(* IEC 61131-3 sources: moqui-plc/iec61131/moqui/framework/src/main/org/moqui/device (part 2) *)

(* ---- ActuatorGroup.st ---- *)
(*
 * ActuatorGroup - demand-driven staging controller for up to ACTUATOR_GROUP_MAX_SIZE on/off actuators.
 *
 * Inspired by ABB ACH580 PFC (Pump and Fan Control, group 76. See ABB ACH580 drive firmware manual).
 * Progressively starts and stops Actuator FBs to match a varying process demand,
 * with automatic priority rotation (autochange) to balance accumulated run hours.
 *
 * Interface with Actuator FBs
 * The caller declares enableRequests and disableRequests arrays and wires them
 * to the VAR_IN_OUT inputs of each Actuator FB:
 *
 *   pump[i](enableRequest := enReq[i], disableRequest := disReq[i], ...);
 *   grp(enableRequests := enReq, disableRequests := disReq, ...);
 *
 * Both the Actuator and ActuatorGroup share the same array by reference (VAR_IN_OUT).
 * ActuatorGroup writes TRUE to issue a command;
 * the Actuator clears the flag to FALSE as its handshake acknowledgment.
 *
 * IMPORTANT: call each Actuator BEFORE ActuatorGroup in the PLC task so that
 * the actuatorEnabled feedback is current when ActuatorGroup evaluates it.
 *
 * Start / stop staging
 * startPoints[k] (k = 0..actuatorNum-1):
 *   While k actuators are running, if demandSetpoint > startPoints[k] continuously
 *   for startDelay, the next available actuator in the priority order is started (subject to runningNum < maxRunning).
 *   startPoints[0] is the threshold to start the very first actuator (0 -> 1).
 *
 * stopPoints[k] (k = 0..actuatorNum-2):
 *   While k+1 actuators are running, if demandSetpoint < stopPoints[k] continuously
 *   for stopDelay, the lowest-priority running actuator is stopped (subject to runningNum > minRunning).
 *   stopPoints[0] is the threshold to stop the last remaining actuator (1 -> 0).
 *
 * Demand must hold on one side of the threshold for the full delay before any action is taken.
 * Crossing back resets the timer (anti-cycling hysteresis).
 *
 * Fault / interlock recovery:
 *   Faulted or interlocked actuators are skipped during start selection.
 *   If a running actuator faults and runningNum drops below minRunning, the next
 *   available standby is started immediately (without waiting for startDelay).
 *
 * Autochange:
 * EvenWear: Rotate when the run-hour gap between any two non-faulted
 *           actuators exceeds maxWearImbalance AND demand <= autochangeLevel.
 *           The priority array is re-sorted by ascending runHours every cycle;
 *           a physical swap (stop most-used, start least-used) is
 *           triggered only when the imbalance threshold is exceeded.
 * FixedInterval: Rotate every autochangeInterval when demand <= autochangeLevel.
 * ExternalTrigger: Rotate on a rising edge of autochangeTrigger when demand <= autochangeLevel.
 * AllStopped: Rotate the index array whenever all actuators stop (group
 *             transitions to Disabled). No physical swap is needed because
 *             all are already stopped; the new order takes effect at the next group enable.
 *
 * Rotation sequence (EvenWear / FixedInterval / ExternalTrigger):
 *   1. Stop the selected actuator (disableRequest).
 *   2. Update the priority array (rotate or re-sort).
 *   3. Start the new highest-priority standby actuator (enableRequest).
 *   The group is in the Autochange FSM state for the duration of this sequence.
 *   runningNum briefly drops by 1; set minRunning = 0 if a momentary reduction
 *   is unacceptable and use process-side redundancy instead.
 *)
FUNCTION_BLOCK ActuatorGroup
	VAR_EXTERNAL CONSTANT
	    (*
		 * Maximum actuators supported. Array bounds in VAR_IN_OUT / VAR_INPUT
	     * must match this size exactly in the caller's declaration.
		 *)
	    ACTUATOR_GROUP_MAX_SIZE : UINT;
	END_VAR
	VAR_IN_OUT
	    (*
	     * Handshake arrays shared with the individual Actuator FBs.
	     * ActuatorGroup writes TRUE to command a start or stop.
	     * Each Actuator FB clears the flag to FALSE when it accepts the command.
	     *)
	    enableRequests : ARRAY[1..ACTUATOR_GROUP_MAX_SIZE] OF BOOL;
	    disableRequests : ARRAY[1..ACTUATOR_GROUP_MAX_SIZE] OF BOOL;
	END_VAR
	VAR_INPUT
		(* Actuator group metadata for logging purpose *)
		actuatorGroupId : STRING;
		actuatorGroupName : STRING;

	    (* Topology *)
	    (* Total actuators declared in the group. Must be 1..ACTUATOR_GROUP_MAX_SIZE. *)
	    actuatorNum : UINT := 1;
	    (* Minimum actuators to keep running simultaneously (0 = allow full stop). *)
	    minRunning : UINT := 1;
	    (* Maximum actuators allowed running simultaneously. *)
	    maxRunning : UINT := 1;

	    (* Process demand *)
	    (* Demand setpoint in percent (0.0 ... 100.0). Drives all start/stop decisions. *)
	    demandSetpoint : REAL;

	    (*
	     * Start / stop thresholds.
	     * startPoints[k]: demand level that triggers starting the (k+1)-th
	     * actuator while exactly k are currently running (k = 0..actuatorNum-1).
	     * startPoints[0] = threshold to start the first actuator (0 -> 1).
		 *)
	    startPoints : ARRAY[0..7] OF REAL;
	    (*
	     * stopPoints[k]: demand level below which the (k+1)-th running actuator is stopped (k = 0..actuatorNum-2).
	     * stopPoints[0] = threshold to stop the last actuator (1 -> 0).
	     *)
	    stopPoints : ARRAY[0..7] OF REAL;
	    (* Demand must stay above startPoints[k] for this long before a start. *)
	    startDelay : TIME := T#10s;
	    (* Demand must stay below stopPoints[k] for this long before a stop. *)
	    stopDelay : TIME := T#10s;

	    (* Autochange *)
	    autochange : ActuatorGroupAutochange := ActuatorGroupAutochange.None;
	    (* Period for FixedInterval rotation. *)
	    autochangeInterval : TIME := T#1h;
	    (*
	     * Max allowed run-hour gap between most-used and least-used actuator
	     * before EvenWear triggers a swap (hours, e.g. 72.0 for 3 days).
	     *)
	    maxWearImbalance : REAL := 72.0;
	    (* Autochange is only triggered when demandSignal <= autochangeLevel. *)
	    autochangeLevel : REAL := 100.0;
	    (* Rising edge triggers an immediate autochange (ExternalTrigger mode). *)
	    autochangeTrigger : BOOL;

	    (* Per-actuator feedback *)
	    (*
	     * Map actuatorEnabled[i] from Actuator[i].enable (TRUE in EnablePhase
	     * AND Enabled states - i.e., the actuator is active or starting up).
	     *)
	    actuatorEnabled : ARRAY[1..ACTUATOR_GROUP_MAX_SIZE] OF BOOL;
	    (* Map actuatorFault[i] from Actuator[i].fault. *)
	    actuatorFault : ARRAY[1..ACTUATOR_GROUP_MAX_SIZE] OF BOOL;
	    (* External maintenance / hardware interlock flag per actuator. *)
	    actuatorInterlocked : ARRAY[1..ACTUATOR_GROUP_MAX_SIZE] OF BOOL;
	    (* Cumulative run time in hours, maintained by the caller (e.g., a REAL counter incremented by 1/3600 each second). *)
	    runHours : ARRAY[1..ACTUATOR_GROUP_MAX_SIZE] OF REAL;

	    (* Group commands *)
	    (*
	      * Rising edge (FALSE->TRUE) starts the group (Disabled -> Running).
	      * Cleared by the FB when the transition is accepted.
	     *)
	    groupEnable : BOOL;
	    (*
	     * Rising edge (FALSE->TRUE) stops the group (Running -> Stopping -> Disabled).
	     * Cleared by the FB when the transition is accepted.
	     *)
	    groupDisable : BOOL;
	END_VAR
	VAR_OUTPUT
	    (* Current group FSM state. *)
	    status : ActuatorGroupStatus := ActuatorGroupStatus.Disabled;
	    (* Actuators neither faulted nor interlocked (available for use). *)
	    availableNum : UINT;
	    (* Actuators currently active (Enabled or EnablePhase). *)
	    runningNum : UINT;
	    (* TRUE when nAvailable < actuatorNum (one or more offline/faulted). *)
	    degraded : BOOL;
	    (* TRUE when a fault has left runningNum below minRunning. *)
	    underMinimum : BOOL;
	    (* TRUE when configuration inputs are invalid. *)
	    invalidConfig : BOOL;
	    (* TRUE while an autochange rotation is in progress. *)
	    autochangeActive : BOOL;
		(* Logger name for centralized signal management *)
		loggerName : STRING;
	END_VAR
	VAR
	    (* Internal FSM state *)
	    internalStatus : ActuatorGroupStatus := ActuatorGroupStatus.Disabled;

	    (* Priority order *)
	    (*
		 * sortedIdx[1] = first to start / last to stop.
	     * sortedIdx[actuatorNum] = last to start / first to stop.
	     * Initialised to [1, 2, … actuatorNum] on the first call.
	     *)
	    sortedIdx : ARRAY[1..ACTUATOR_GROUP_MAX_SIZE] OF UINT;

	    (* Autochange bookkeeping *)
	    autochangeStep : UINT; (* 0 = idle, 1 = stopping old, 2 = starting new *)
	    autochangeStopIdx : UINT; (* physical actuator slot being stopped *)
	    autochangeStartIdx : UINT; (* physical actuator slot being started *)
	    autochangeTrigOld : BOOL; (* previous cycle value for edge detection *)

	    (* Timer signals *)
	    (* Computed each cycle in the FSM; passed to TON FBs at the bottom. *)
	    startTimerTrig : BOOL;
	    stopTimerTrig : BOOL;
	    autochangeTimerTrig : BOOL;
	    startTimer : TON;
	    stopTimer : TON;
	    autochangeTimer : TON;

	    (* Loop temporaries *)
	    i, j, tempIdx : UINT;
	    swapped : BOOL;
	    minHoursIdx : UINT;
	    maxHoursIdx : UINT;
		(* Logger facade *)
		logger : LoggerFacade;
		init : BOOL;
	END_VAR

	(* Init *)
	IF NOT init THEN
		IF (actuatorGroupId = '' AND actuatorGroupName = '') THEN
			invalidConfig := TRUE;
			RETURN;
		END_IF;

		(* Logger facade init *)
		loggerName := concat(concat(concat(actuatorGroupName, '['), actuatorGroupId), ']');
		logger.enable := TRUE; logger.loggerName := loggerName;
		init := TRUE;
	END_IF;

	logger(message := 'Running actuator group.', level := LogLevel.DEBUG);

	(* Args validation *)
	invalidConfig := (actuatorNum < 1) OR (actuatorNum > ACTUATOR_GROUP_MAX_SIZE)
		OR (minRunning < 0) OR (maxRunning < 1)
	    OR (minRunning > maxRunning)
	    OR (maxRunning > actuatorNum);
	IF invalidConfig THEN
	    status := ActuatorGroupStatus.Disabled;
	    RETURN;
	END_IF;

	(* Init priority index on first call or when actuatorNum grows.
	 * Valid slot indices are 1..actuatorNum; 0 is the zero-initialised
	 * default and is never a valid value, so a zero entry always means the slot
	 * has not been assigned yet. This allows the group to be reconfigured at
	 * run-time with a larger actuatorNum without re-setting existing order. *)
	FOR i := 1 TO actuatorNum DO
	    IF sortedIdx[i] = 0 THEN
	        sortedIdx[i] := i;
	    END_IF;
	END_FOR;

	(* Count available and active actuators (every cycle) *)
	availableNum := 0;
	runningNum   := 0;
	FOR i := 1 TO actuatorNum DO
	    IF NOT actuatorFault[i] AND NOT actuatorInterlocked[i] THEN
	        availableNum := availableNum + 1;
	    END_IF;
	    IF actuatorEnabled[i] THEN
	        runningNum := runningNum + 1;
	    END_IF;
	END_FOR;
	degraded := (availableNum < actuatorNum);
	underMinimum := (internalStatus = ActuatorGroupStatus.Running) AND (runningNum < minRunning);

	(* EvenWear priority re-sort (runs every cycle when EvenWear is active) *)
	(*
	 * Sort sortedIdx[1..actuatorNum] by ascending runHours so that the actuator
	 * with the fewest cumulative hours is always started first.
	 * Faulted / interlocked actuators are bubbled to the end of the array so they
	 * are naturally skipped when the start/stop logic scans the priority order.
	 *
	 * The sort runs every cycle in Running and Autochange states.  For other
	 * autochange modes the order is updated only by explicit rotation steps.
	 *)
	IF autochange = ActuatorGroupAutochange.EvenWear
	        AND (internalStatus = ActuatorGroupStatus.Running
			OR internalStatus = ActuatorGroupStatus.Autochange) THEN
	    FOR i := 1 TO actuatorNum - 1 DO
	        swapped := FALSE;
	        FOR j := 1 TO actuatorNum - i DO
	            (* Push faulted / interlocked slots to the end *)
	            IF (actuatorFault[sortedIdx[j]] OR actuatorInterlocked[sortedIdx[j]])
	                    AND NOT (actuatorFault[sortedIdx[j + 1]] OR actuatorInterlocked[sortedIdx[j + 1]])
	               (* Among healthy slots: sort by ascending run hours *)
	               OR (NOT (actuatorFault[sortedIdx[j]] OR actuatorInterlocked[sortedIdx[j]])
	                   AND NOT (actuatorFault[sortedIdx[j + 1]] OR actuatorInterlocked[sortedIdx[j + 1]])
	                   AND runHours[sortedIdx[j]] > runHours[sortedIdx[j + 1]]) THEN
	                tempIdx := sortedIdx[j];
	                sortedIdx[j] := sortedIdx[j + 1];
	                sortedIdx[j + 1] := tempIdx;
	                swapped := TRUE;
	            END_IF;
	        END_FOR;

	        IF NOT swapped THEN EXIT; END_IF;
	    END_FOR;
	END_IF;

	(* Timer signal defaults (overridden by the Running state block) *)
	startTimerTrig := FALSE;
	stopTimerTrig := FALSE;
	(*
	 * AutochangeTimer only accumulates while Running - interval is operating time, not wall time.
	 * The Running state sets this FALSE for one cycle after .Q fires to reset the period.
	 *)
	autochangeTimerTrig := (autochange = ActuatorGroupAutochange.FixedInterval)
		AND (internalStatus = ActuatorGroupStatus.Running);

	(* Main FSM *)
	CASE internalStatus OF
	    (* Disabled: no actuators running. Wait for groupEnable. *)
	    ActuatorGroupStatus.Disabled :
	        groupDisable := FALSE;
	        autochangeActive := FALSE;
	        autochangeStep := 0;

	        IF groupEnable AND availableNum >= minRunning THEN
				logger(message := 'Actuator group running.', level := LogLevel.DEBUG);
	            groupEnable := FALSE;
	            internalStatus := ActuatorGroupStatus.Running;
	        ELSIF groupEnable AND availableNum < minRunning THEN
	            (* Not enough actuators available - refuse enable *)
	            groupEnable := FALSE;
	        END_IF;

	    (* Running: demand-driven start / stop of individual actuators. *)
	    ActuatorGroupStatus.Running :
	        groupEnable := FALSE;
	        autochangeActive := FALSE;

	        (* Disable command: transition to Stopping *)
	        IF groupDisable THEN
	            groupDisable := FALSE;
	            FOR i := 1 TO actuatorNum DO
	                IF actuatorEnabled[i] THEN
	                    disableRequests[i] := TRUE;
	                END_IF;
	                enableRequests[i] := FALSE; (* Cancel pending starts *)
	            END_FOR;

				internalStatus := ActuatorGroupStatus.Stopping;
				logger(message := 'Actuator group stopping.', level := LogLevel.DEBUG);
	        ELSE
	            (* Fault recovery: restore minRunning immediately (no delay). *)
	            (*
	             * If a running actuator has faulted and runningNum < minRunning,
	             * start the next available standby without waiting for startDelay.
	             * Only one start per cycle to avoid over-driving the process.
	             *)
	            IF runningNum < minRunning THEN
	                FOR i := 1 TO actuatorNum DO
	                    IF NOT actuatorEnabled[sortedIdx[i]]
								AND NOT actuatorFault[sortedIdx[i]]
	                            AND NOT actuatorInterlocked[sortedIdx[i]]
	                            AND NOT enableRequests[sortedIdx[i]] THEN
	                        enableRequests[sortedIdx[i]] := TRUE;
	                        EXIT;
	                    END_IF;
	                END_FOR;
	            END_IF;

	            (* Normal start: add the next unit when demand is high. *)
	            (*
	             * Check startPoints[runningNum]: the threshold to go from runningNum to runningNum+1 active actuators.
				 * Array index matches the current running count (ABB 76.30: "velocity to start auxiliary k").
	             * The timer runs as long as the condition holds; it resets
	             * automatically if demand drops back below the threshold.
	             *)
	            IF runningNum >= minRunning AND runningNum < maxRunning
	                    AND runningNum <= actuatorNum - 1 THEN
	                startTimerTrig := (demandSetpoint > startPoints[runningNum]);
	                IF startTimer.Q THEN
	                    FOR i := 1 TO actuatorNum DO
	                        IF NOT actuatorEnabled[sortedIdx[i]]
	                                AND NOT actuatorFault[sortedIdx[i]]
	                                AND NOT actuatorInterlocked[sortedIdx[i]]
	                                AND NOT enableRequests[sortedIdx[i]] THEN
	                            enableRequests[sortedIdx[i]] := TRUE;
	                            EXIT;
	                        END_IF;
	                    END_FOR;

	                    startTimerTrig := FALSE; (* Reset timer after issuing start *)
	                END_IF;
	            END_IF;

	            (* Normal stop: remove the last unit when demand is low. *)
	            (*
	             * Check stopPoints[runningNum - 1]: the threshold to go from runningNum
	             * to runningNum-1 active actuators. Index runningNum-1 is always >= 0
	             * because runningNum > minRunning >= 0. The last actuator in the
	             * sorted order (highest index) is stopped first (LIFO principle).
	             *)
	            IF runningNum > minRunning
	                    AND runningNum - 1 <= actuatorNum - 1 THEN
	                stopTimerTrig := (demandSetpoint < stopPoints[runningNum - 1]);
	                IF stopTimer.Q THEN
	                    FOR i := actuatorNum TO 1 BY -1 DO
	                        IF actuatorEnabled[sortedIdx[i]]
	                                AND NOT disableRequests[sortedIdx[i]] THEN
	                            disableRequests[sortedIdx[i]] := TRUE;
	                            EXIT;
	                        END_IF;
	                    END_FOR;

	                    stopTimerTrig := FALSE; (* Reset timer after issuing stop *)
	                END_IF;
	            END_IF;

	            (* Autochange trigger evaluation *)
	            IF autochange <> ActuatorGroupAutochange.None
	                    AND autochange <> ActuatorGroupAutochange.AllStopped
	                    AND runningNum > 0
	                    AND demandSetpoint <= autochangeLevel THEN

	                CASE autochange OF
	                    (* EvenWear *)
	                    ActuatorGroupAutochange.EvenWear :
	                        (*
	                         * Find the running actuator with the most hours and the
	                         * standby actuator with the fewest hours.
							 * Trigger a swap when the imbalance exceeds maxWearImbalance (hours).
	                         *)
	                        minHoursIdx := 0; maxHoursIdx := 0;
	                        FOR i := 1 TO actuatorNum DO
	                            IF NOT actuatorFault[i] AND NOT actuatorInterlocked[i] THEN
	                                IF minHoursIdx = 0 THEN
	                                    minHoursIdx := i;
	                                ELSIF runHours[i] < runHours[minHoursIdx] THEN
	                                    minHoursIdx := i;
	                                END_IF;
	                                IF maxHoursIdx = 0 THEN
	                                    maxHoursIdx := i;
	                                ELSIF runHours[i] > runHours[maxHoursIdx] THEN
	                                    maxHoursIdx := i;
	                                END_IF;
	                            END_IF;
	                        END_FOR;

	                        IF minHoursIdx > 0 AND maxHoursIdx > 0
	                                AND minHoursIdx <> maxHoursIdx
	                                AND (runHours[maxHoursIdx] - runHours[minHoursIdx]) > maxWearImbalance
	                                AND actuatorEnabled[maxHoursIdx]
	                                AND NOT actuatorEnabled[minHoursIdx]
	                                AND NOT actuatorFault[minHoursIdx]
	                                AND NOT actuatorInterlocked[minHoursIdx] THEN
	                            autochangeStopIdx := maxHoursIdx;
	                            autochangeStartIdx := 0; (* Resolved in Autochange step 1 *)
	                            autochangeStep := 1;
	                            disableRequests[autochangeStopIdx] := TRUE;
	                            internalStatus := ActuatorGroupStatus.Autochange;
	                        END_IF;

	                    (* FixedInterval *)
	                    ActuatorGroupAutochange.FixedInterval :
	                        IF autochangeTimer.Q THEN
	                            (* Select the lowest-priority running actuator to stop *)
	                            autochangeStopIdx := 0;
	                            FOR i := actuatorNum TO 1 BY -1 DO
	                                IF actuatorEnabled[sortedIdx[i]] THEN
	                                    autochangeStopIdx := sortedIdx[i];
	                                    EXIT;
	                                END_IF;
	                            END_FOR;

	                            IF autochangeStopIdx > 0 THEN
	                                autochangeStep := 1;
	                                disableRequests[autochangeStopIdx] := TRUE;
	                                internalStatus := ActuatorGroupStatus.Autochange;
	                            END_IF;

	                            (* Reset the interval timer regardless of whether we swapped *)
	                            autochangeTimerTrig := FALSE;
	                        END_IF;

	                    (* ExternalTrigger *)
	                    ActuatorGroupAutochange.ExternalTrigger :
	                        IF autochangeTrigger AND NOT autochangeTrigOld THEN
	                            autochangeStopIdx := 0;

	                            FOR i := actuatorNum TO 1 BY -1 DO
	                                IF actuatorEnabled[sortedIdx[i]] THEN
	                                    autochangeStopIdx := sortedIdx[i];
	                                    EXIT;
	                                END_IF;
	                            END_FOR;

	                            IF autochangeStopIdx > 0 THEN
	                                autochangeStep := 1;
	                                disableRequests[autochangeStopIdx] := TRUE;
	                                internalStatus := ActuatorGroupStatus.Autochange;
	                            END_IF;
	                        END_IF;
	                END_CASE;
	            END_IF;
	        END_IF; (* groupDisable / else *)

	    (* Stopping: wait for all actuators to reach disabled state. *)
	    ActuatorGroupStatus.Stopping :
	        IF runningNum = 0 THEN
	            (*
	             * AllStopped autochange: rotate the priority order now that all
	             * actuators are off.  The new order takes effect at the next
	             * groupEnable.  No physical swap is needed (all already stopped).
	             *)
	            IF autochange = ActuatorGroupAutochange.AllStopped THEN
	                tempIdx := sortedIdx[1];
	                FOR i := 1 TO actuatorNum - 1 DO
	                    sortedIdx[i] := sortedIdx[i + 1];
	                END_FOR;
	                sortedIdx[actuatorNum] := tempIdx;
	            END_IF;

	            internalStatus := ActuatorGroupStatus.Disabled;
	        END_IF;

	    (*
	     * Autochange: sequential stop / rotate / start.
	     *
	     * Step 1 - wait for the old actuator to stop.
	     * Step 2 - start the new highest-priority standby.
	     *)
	    ActuatorGroupStatus.Autochange :
			logger(message := 'Actuator group autochange.', level := LogLevel.DEBUG);
	        autochangeActive := TRUE;
	        groupEnable := FALSE;

	        (* Disable command during autochange: abort and go to Stopping *)
	        IF groupDisable THEN
	            groupDisable := FALSE;

	            FOR i := 1 TO actuatorNum DO
	                IF actuatorEnabled[i] THEN disableRequests[i] := TRUE; END_IF;
	                enableRequests[i] := FALSE;
	            END_FOR;

	            internalStatus := ActuatorGroupStatus.Stopping;
	        ELSE
	            CASE autochangeStep OF
	                1 : (* Waiting for the old actuator to finish stopping *)
	                    IF NOT actuatorEnabled[autochangeStopIdx] THEN
	                        (*
	                         * Old actuator is now off.  Update the priority order:
	                         * - FixedInterval / ExternalTrigger: rotate the stopped
	                         *   actuator from its current position to the end of the
	                         *   array so it is the last to be started next time.
	                         * - EvenWear: the continuous sort (above) already
	                         *   maintains the correct order; no manual rotation needed.
	                         *)
	                        IF autochange = ActuatorGroupAutochange.FixedInterval
	                                OR autochange = ActuatorGroupAutochange.ExternalTrigger THEN
	                            FOR i := 1 TO actuatorNum DO
	                                IF sortedIdx[i] = autochangeStopIdx THEN
	                                    FOR j := i TO actuatorNum - 1 DO
	                                        sortedIdx[j] := sortedIdx[j + 1];
	                                    END_FOR;
	                                    sortedIdx[actuatorNum] := autochangeStopIdx;
	                                    EXIT;
	                                END_IF;
	                            END_FOR;
	                        END_IF;

	                        (* Find the highest-priority standby to start *)
	                        autochangeStartIdx := 0;
	                        FOR i := 1 TO actuatorNum DO
	                            IF NOT actuatorEnabled[sortedIdx[i]]
	                                    AND NOT actuatorFault[sortedIdx[i]]
	                                    AND NOT actuatorInterlocked[sortedIdx[i]] THEN
	                                autochangeStartIdx := sortedIdx[i];
	                                EXIT;
	                            END_IF;
	                        END_FOR;

	                        IF autochangeStartIdx > 0 THEN
	                            enableRequests[autochangeStartIdx] := TRUE;
	                            autochangeStep := 2;
	                        ELSE
	                            (* No standby available; return without starting a replacement *)
	                            autochangeStep := 0;
	                            internalStatus := ActuatorGroupStatus.Running;
	                        END_IF;
	                    END_IF;

	                2 : (* Waiting for the new actuator to reach enabled state *)
	                    IF actuatorEnabled[autochangeStartIdx] THEN
	                        autochangeStep := 0;
	                        internalStatus := ActuatorGroupStatus.Running;
	                    END_IF;
	            END_CASE;
	        END_IF;
	END_CASE; (* internalStatus *)

	(* Unconditional timer calls (once per cycle, after FSM) *)
	(*
	 * startTimer / stopTimer: anti-cycling guards for demand-driven start/stop.
	 *   IN is driven by the Running state logic above.
	 *   IN goes FALSE automatically when:
	 *     - demand reverses (anti-cycling, timer resets before Q fires), or
	 *     - the FSM exits Running state (timer.IN defaults to FALSE above), or
	 *     - a start/stop action is taken (timer.IN forced FALSE in the action).
	 *
	 * autochangeTimer: fixed-interval rotation period. Runs whenever
	 *   autochange = FixedInterval, regardless of FSM state.  The timer is
	 *   reset by setting autochangeTimer_IN := FALSE for one cycle (done in
	 *   the Running state when the timer fires).
	 *)
	startTimer(IN := startTimerTrig, PT := startDelay);
	stopTimer(IN := stopTimerTrig, PT := stopDelay);
	autochangeTimer(IN := autochangeTimerTrig, PT := autochangeInterval);

	(* Rising-edge latch - update after all logic that reads it *)
	autochangeTrigOld := autochangeTrigger;

	(* Status output *)
	status := internalStatus;
	END_FUNCTION_BLOCK

(* ---- DeviceConfigCmds.pou ---- *)
(*#-#-#-#-#-#-#-#-#-#---Declaration---#-#-#-#-#-#-#-#-#-#-#-#-#*)

{attribute 'no_assign'}
FUNCTION_BLOCK DeviceConfigCmds
VAR_EXTERNAL CONSTANT
	DEVICE_CONFIG_LIST_MAX_SIZE : UINT;
	defaultConfigType : STRING;
END_VAR
VAR_INPUT
    configType : STRING := defaultConfigType; (* If empty, set default device config type *)
	(*
     * The default file name of a recipe is: <configName>.<configType>.<extension>
     * Device config ID or name used by the commands.
     *)
    configName : STRING := '';
    cmd : DeviceConfigCmdType := DeviceConfigCmdType.Load;
END_VAR
VAR_OUTPUT
	(* Device config list *)
	configNameList : ARRAY[0..DEVICE_CONFIG_LIST_MAX_SIZE] OF STRING;
	configNameListSize : UINT;
	error : BOOL;
	errorId : DWORD; (* 16#5000 : InvalidArgs *)
END_VAR
VAR
	(* Recipe management component *)
    configCmds : Recipe_Management.RecipeManCommands;
	(* Logger facade *)
	logger : LoggerFacade;
    i : UINT;
END_VAR

(*#-#-#-#-#-#-#-#-#-#---Implementation---#-#-#-#-#-#-#-#-#-#-#-#-#*)

IF cmd = DeviceConfigCmdType.Init THEN
	(* Logger facade init *)
	logger.enable := TRUE; logger.loggerName := 'DeviceConfigCmds';
END_IF;

(* Args validation *)
IF (configType = '') OR (cmd <> DeviceConfigCmdType.Init AND cmd <> DeviceConfigCmdType.Reset AND configName = '') THEN
	logger(message := 'Invalid arguments.', level := LogLevel.Error);
	error := TRUE;
	errorId := 16#5000;
	RETURN;
END_IF;

CASE cmd OF
	DeviceConfigCmdType.Init :
		logger(message := 'Loading device config list.');
		(* Clear previous list on reload *)
		FOR i := 0 TO DEVICE_CONFIG_LIST_MAX_SIZE DO configNameList[i] := ''; END_FOR;
		configNameListSize := 0;

		errorId := configCmds.ReloadRecipes(RecipeDefinitionName := configType);
		error := (errorId <> 0);
		IF error THEN logger(message := 'Error loading device config list from file system.', level := LogLevel.Error); RETURN; END_IF;

		(* iSize is the array capacity: DEVICE_CONFIG_LIST_MAX_SIZE + 1 elements (indices 0..MAX) *)
		errorId := configCmds.GetRecipeNames(RecipeDefinitionName := configType,
			pStrings := ADR(configNameList), iSize := TO_INT(DEVICE_CONFIG_LIST_MAX_SIZE) + 1, iStartIndex := 0);
		error := (errorId <> 0);
		IF error THEN logger(message := 'Error loading device config names.', level := LogLevel.Error); RETURN; END_IF;
		(* Set the actual number of recipes/device configs found *)
		configNameListSize := TO_UINT(MIN(configCmds.GetRecipeCount(RecipeDefinitionName := configType),
			TO_DINT(DEVICE_CONFIG_LIST_MAX_SIZE) + 1));

    DeviceConfigCmdType.Create :
		errorId := configCmds.CreateRecipe(RecipeDefinitionName := configType, RecipeName := configName);
        error := (errorId <> 0);
		IF error THEN
			logger(message := concat(concat(concat('Error creating device config ', configName), ' of type '), configType), level := LogLevel.Error);
		ELSE
			logger(message := concat(concat(concat('Created device config ', configName), ' of type '), configType));
        END_IF;

    DeviceConfigCmdType.Save :
        errorId := configCmds.ReadAndSaveRecipe(RecipeDefinitionName := configType, RecipeName := configName);
        error := (errorId <> 0);
        IF error THEN
			logger(message := concat(concat(concat('Error saving device config ', configName), ' of type '), configType), level := LogLevel.Error);
		ELSE
           	logger(message := concat(concat(concat('Saved device config ', configName), ' of type '), configType));
		END_IF;

	DeviceConfigCmdType.Load:
        errorId := configCmds.LoadAndWriteRecipe(RecipeDefinitionName := configType, RecipeName := configName);
        error := (errorId <> 0);
		IF error THEN
			logger(message := concat(concat(concat('Error loading device config ', configName), ' of type '), configType), level := LogLevel.Error);
		ELSE
        	logger(message := concat(concat(concat('Loaded device config ', configName), ' of type '), configType));
        END_IF;

    DeviceConfigCmdType.Delete:
        errorId := configCmds.DeleteRecipeFile(RecipeDefinitionName := configType, RecipeName := configName);
		error := (errorId <> 0);
		IF error THEN
			logger(message := concat('Error deleting file for device config ', configName), level := LogLevel.Error);
			RETURN;
		END_IF;

		errorId := configCmds.DeleteRecipe(RecipeDefinitionName := configType, RecipeName := configName);
        error := (errorId <> 0);
        IF error THEN
			logger(message := concat(concat(concat('Error deleting device config ', configName), ' of type '), configType), level := LogLevel.Error);
		ELSE
			logger(message := concat(concat(concat('Deleted device config ', configName), ' of type '), configType));
        END_IF;

	DeviceConfigCmdType.Reset :
		logger(message := 'Resetting device config list.');
		configCmds.ResetLastError();
		configCmds.ResetLastInfo();
		error := FALSE;
		errorId := 0;
END_CASE;

(* ---- DeviceConfigCmds.st ---- *)
FUNCTION_BLOCK DeviceConfigCmds
	VAR_EXTERNAL CONSTANT
		DEVICE_CONFIG_LIST_MAX_SIZE : UINT;
		defaultConfigType : STRING;
		deviceConfigStoragePath : STRING;
	END_VAR
	VAR_INPUT
	    configType : STRING := defaultConfigType; (* If empty, set default device config type *)
		(*
	     * The default file name of a recipe is: <configName>.<configType>.<extension>
	     * Device config ID or name used by the commands.
	     *)
	    configName : STRING := '';
	    cmd : DeviceConfigCmdType := DeviceConfigCmdType.Load;
	END_VAR
	VAR_OUTPUT
		(* Device config list *)
		configNameList : ARRAY[0..DEVICE_CONFIG_LIST_MAX_SIZE] OF STRING;
		configNameListSize : UINT;
		error : BOOL;
		errorId : DWORD; (* 16#5000 : InvalidArgs *)
	END_VAR
	VAR
		(* Recipe management component *)
	    configCmds : Recipe_Management.RecipeManCommands;
		(* Logger facade *)
		logger : LoggerFacade;
	    i, j : UINT;
		sortTemp : STRING; sortSwapped : BOOL;
	END_VAR

	IF cmd = DeviceConfigCmdType.Init THEN
		(* Logger facade init *)
		logger.enable := TRUE; logger.loggerName := 'DeviceConfigCmds';
	END_IF;

	(* Args validation *)
	IF (configType = '') OR (cmd <> DeviceConfigCmdType.Init AND cmd <> DeviceConfigCmdType.Reset AND configName = '') THEN
		logger(message := 'Invalid arguments.', level := LogLevel.Error);
		error := TRUE;
		errorId := 16#5000;
		RETURN;
	END_IF;

	CASE cmd OF
		DeviceConfigCmdType.Init :
			logger(message := 'Loading device config list.');
			(* Clear previous list on reload *)
			FOR i := 0 TO DEVICE_CONFIG_LIST_MAX_SIZE DO configNameList[i] := ''; END_FOR;
			configNameListSize := 0;

			IF deviceConfigStoragePath <> '' THEN
				configCmds.SetStoragePath(stPath := deviceConfigStoragePath);
			END_IF;
			errorId := configCmds.ReloadRecipes(RecipeDefinitionName := configType);
			error := (errorId <> 0);
			IF error THEN logger(message := 'Error loading device config list from file system.', level := LogLevel.Error); RETURN; END_IF;

			(* iSize is the array capacity: DEVICE_CONFIG_LIST_MAX_SIZE + 1 elements (indices 0..MAX) *)
			errorId := configCmds.GetRecipeNames(RecipeDefinitionName := configType,
				pStrings := ADR(configNameList), iSize := TO_INT(DEVICE_CONFIG_LIST_MAX_SIZE) + 1, iStartIndex := 0);
			error := (errorId <> 0);
			IF error THEN logger(message := 'Error loading device config names.', level := LogLevel.Error); RETURN; END_IF;
			(* Set the actual number of recipes/device configs found *)
			configNameListSize := TO_UINT(MIN(configCmds.GetRecipeCount(RecipeDefinitionName := configType),
				TO_DINT(DEVICE_CONFIG_LIST_MAX_SIZE) + 1));

			(* Sort recipe names alphabetically (ascending bubble sort) *)
			IF configNameListSize > 1 THEN
				REPEAT
					sortSwapped := FALSE;
					FOR j := 0 TO configNameListSize - 2 DO
						IF configNameList[j] > configNameList[j + 1] THEN
							sortTemp := configNameList[j];
							configNameList[j] := configNameList[j + 1];
							configNameList[j + 1] := sortTemp;
							sortSwapped := TRUE;
						END_IF;
					END_FOR;
				UNTIL NOT sortSwapped
				END_REPEAT;
			END_IF;

	    DeviceConfigCmdType.Create :
			errorId := configCmds.CreateRecipe(RecipeDefinitionName := configType, RecipeName := configName);
	        error := (errorId <> 0);
			IF error THEN
				logger(message := concat(concat(concat('Error creating device config ', configName), ' of type '), configType), level := LogLevel.Error);
			ELSE
				logger(message := concat(concat(concat('Created device config ', configName), ' of type '), configType));
	        END_IF;

	    DeviceConfigCmdType.Save :
	        errorId := configCmds.ReadAndSaveRecipe(RecipeDefinitionName := configType, RecipeName := configName);
	        error := (errorId <> 0);
	        IF error THEN
				logger(message := concat(concat(concat('Error saving device config ', configName), ' of type '), configType), level := LogLevel.Error);
			ELSE
	           	logger(message := concat(concat(concat('Saved device config ', configName), ' of type '), configType));
			END_IF;

		DeviceConfigCmdType.Load:
	        errorId := configCmds.LoadAndWriteRecipe(RecipeDefinitionName := configType, RecipeName := configName);
	        error := (errorId <> 0);
			IF error THEN
				logger(message := concat(concat(concat('Error loading device config ', configName), ' of type '), configType), level := LogLevel.Error);
			ELSE
	        	logger(message := concat(concat(concat('Loaded device config ', configName), ' of type '), configType));
	        END_IF;

	    DeviceConfigCmdType.Delete:
	        errorId := configCmds.DeleteRecipeFile(RecipeDefinitionName := configType, RecipeName := configName);
			error := (errorId <> 0);
			IF error THEN
				logger(message := concat('Error deleting file for device config ', configName), level := LogLevel.Error);
				RETURN;
			END_IF;

			errorId := configCmds.DeleteRecipe(RecipeDefinitionName := configType, RecipeName := configName);
	        error := (errorId <> 0);
	        IF error THEN
				logger(message := concat(concat(concat('Error deleting device config ', configName), ' of type '), configType), level := LogLevel.Error);
			ELSE
				logger(message := concat(concat(concat('Deleted device config ', configName), ' of type '), configType));
	        END_IF;

		DeviceConfigCmdType.Reset :
			logger(message := 'Resetting device config list.');
			configCmds.ResetLastError();
			configCmds.ResetLastInfo();
			error := FALSE;
			errorId := 0;
	END_CASE;
	END_FUNCTION_BLOCK

(* ---- DeviceConfigMgmt.pou ---- *)
(*#-#-#-#-#-#-#-#-#-#---Declaration---#-#-#-#-#-#-#-#-#-#-#-#-#*)

{attribute 'no_assign'}
(*
 * Pure recipe sequencing logic. Implement complex logic, including micro-recipe composition,
 * alternative recipes, condition-based recipes, etc., if needed.
 *)
FUNCTION_BLOCK DeviceConfigMgmt
VAR_EXTERNAL CONSTANT
	defaultConfigType : STRING;
END_VAR
VAR_INPUT
	enable : BOOL;
	continueAfterError : BOOL;
	configCompleted : BOOL; (* Config processed feedback *)
END_VAR
VAR_OUTPUT
    done, allConfigLoaded, busy, error : BOOL;
	errorId : DWORD;
END_VAR
VAR
    status : DeviceConfigMgmtStatus := DeviceConfigMgmtStatus.Idle;
    configCmds : DeviceConfigCmds;
    currentConfigIndex : UINT := 0;
	(* Logger facade *)
    logger : LoggerFacade;
	init : BOOL;
END_VAR

(*#-#-#-#-#-#-#-#-#-#---Implementation---#-#-#-#-#-#-#-#-#-#-#-#-#*)

IF NOT init THEN
	(* Logger facade init *)
	logger.enable := TRUE; logger.loggerName := 'DeviceConfigMgmt';
	init := TRUE;
END_IF;

CASE status OF
    DeviceConfigMgmtStatus.Idle :
		done := FALSE; busy := FALSE;

        IF enable THEN
			busy := TRUE;
			(* Setup the default config type *)
            configCmds.configType := defaultConfigType;
            status := DeviceConfigMgmtStatus.Init;
        END_IF;

    DeviceConfigMgmtStatus.Init :
		allConfigLoaded := FALSE;
		configCmds(cmd := DeviceConfigCmdType.Init, error => error, errorId => errorId);

        IF configCmds.error THEN
			status := DeviceConfigMgmtStatus.Resetting;
		ELSE
            status := DeviceConfigMgmtStatus.Load;
        END_IF;

    DeviceConfigMgmtStatus.Load :
        IF (currentConfigIndex >= configCmds.configNameListSize) THEN
            status := DeviceConfigMgmtStatus.Completed;
        ELSE
            configCmds.configName := configCmds.configNameList[currentConfigIndex];
            configCmds(cmd := DeviceConfigCmdType.Load, error => error, errorId => errorId);
            IF configCmds.error THEN
                status := DeviceConfigMgmtStatus.Resetting;
            ELSE
                status := DeviceConfigMgmtStatus.WaitProcessing;
            END_IF;
        END_IF;

    DeviceConfigMgmtStatus.WaitProcessing :
		done := TRUE;
		busy := FALSE;

        IF configCompleted THEN
            done := FALSE;
            logger(message := concat(concat('Device config ', configCmds.configName), ' completed.'));
            currentConfigIndex := currentConfigIndex + 1;
            status := DeviceConfigMgmtStatus.Load;
        END_IF;

    DeviceConfigMgmtStatus.Completed :
        allConfigLoaded := TRUE;
		done := TRUE;
		busy := FALSE;
		error := FALSE;
		currentConfigIndex := 0;
        logger(message := 'All device configs loaded.');
        status := DeviceConfigMgmtStatus.Idle;

    DeviceConfigMgmtStatus.Resetting :
        configCmds(cmd := DeviceConfigCmdType.Reset, error => error, errorId => errorId);
		IF NOT continueAfterError THEN
        	currentConfigIndex := 0;
        END_IF;

        status := DeviceConfigMgmtStatus.Init;
END_CASE;

(* ---- DeviceConfigMgmt.st ---- *)
(*
 * Pure recipe sequencing logic. Implement complex logic, including micro-recipe composition,
 * alternative recipes, condition-based recipes, etc., if needed.
 *)
FUNCTION_BLOCK DeviceConfigMgmt
	VAR_EXTERNAL CONSTANT
		defaultConfigType : STRING;
	END_VAR
	VAR_INPUT
		enable : BOOL;
		continueAfterError : BOOL;
		configCompleted : BOOL; (* Config processed feedback *)
	END_VAR
	VAR_OUTPUT
	    done, allConfigLoaded, busy, error : BOOL;
		errorId : DWORD;
	END_VAR
	VAR
	    status : DeviceConfigMgmtStatus := DeviceConfigMgmtStatus.Idle;
	    configCmds : DeviceConfigCmds;
	    currentConfigIndex : UINT := 0;
		(* Logger facade *)
	    logger : LoggerFacade;
		init : BOOL;
		configCompletedREdge : R_TRIG;
	END_VAR

	IF NOT init THEN
		(* Logger facade init *)
		logger.enable := TRUE; logger.loggerName := 'DeviceConfigMgmt';
		init := TRUE;
	END_IF;

	configCompletedREdge(CLK := configCompleted);

	CASE status OF
	    DeviceConfigMgmtStatus.Idle :
			done := FALSE; busy := FALSE;

	        IF enable THEN
				busy := TRUE;
				(* Setup the default config type *)
	            configCmds.configType := defaultConfigType;
	            status := DeviceConfigMgmtStatus.Init;
	        END_IF;

	    DeviceConfigMgmtStatus.Init :
			allConfigLoaded := FALSE;
			configCmds(cmd := DeviceConfigCmdType.Init, error => error, errorId => errorId);

	        IF configCmds.error THEN
				status := DeviceConfigMgmtStatus.Resetting;
			ELSE
	            status := DeviceConfigMgmtStatus.Load;
	        END_IF;

	    DeviceConfigMgmtStatus.Load :
	        IF (currentConfigIndex >= configCmds.configNameListSize) THEN
	            status := DeviceConfigMgmtStatus.Completed;
	        ELSE
	            configCmds.configName := configCmds.configNameList[currentConfigIndex];
	            configCmds(cmd := DeviceConfigCmdType.Load, error => error, errorId => errorId);
	            IF configCmds.error THEN
	                status := DeviceConfigMgmtStatus.Resetting;
	            ELSE
	                status := DeviceConfigMgmtStatus.WaitProcessing;
	            END_IF;
	        END_IF;

	    DeviceConfigMgmtStatus.WaitProcessing :
			done := TRUE;
			busy := FALSE;

	        IF configCompletedREdge.Q THEN
	            done := FALSE;
	            logger(message := concat(concat('Device config ', configCmds.configName), ' completed.'));
	            currentConfigIndex := currentConfigIndex + 1;
	            status := DeviceConfigMgmtStatus.Load;
	        END_IF;

	    DeviceConfigMgmtStatus.Completed :
	        allConfigLoaded := TRUE;
			done := TRUE;
			busy := FALSE;
			error := FALSE;
			currentConfigIndex := 0;
	        logger(message := 'All device configs loaded.');
	        status := DeviceConfigMgmtStatus.Idle;

	    DeviceConfigMgmtStatus.Resetting :
	        configCmds(cmd := DeviceConfigCmdType.Reset, error => error, errorId => errorId);
			IF NOT continueAfterError THEN
	        	currentConfigIndex := 0;
	        END_IF;

	        status := DeviceConfigMgmtStatus.Init;
	END_CASE;
	END_FUNCTION_BLOCK

(* ---- EdgeTrigStatusMgr.pou ---- *)
(*#-#-#-#-#-#-#-#-#-#---Declaration---#-#-#-#-#-#-#-#-#-#-#-#-#*)

{attribute 'no_assign'}
(*
Edge triggered status manager.
The PLCOpen standard presents “service/command” function block patterns
that manage the execution of a request (edge-triggered)
or the maintenance of a condition (level-controlled).
The PLCopen patterns model the lifecycle of a command, not the state of the device.
A command handler FB uses the PLCopen (Action) pattern.
The device model maintains the bistable state (Reality/Feedback).
The command requests a device transition, but does not define the device state.
It makes sense to model triggers and levels for physical devices only as an interface contract
between the caller and the device controller, not as the “physical truth” of the device.
An example of edge-triggered functionality is a move-to-position command which,
after being initialized via the input execute, runs till finalized.
For the detection of a rising edge in a function block, two PLC cycles are necessary.
Thus, if the requirement is to be able to process a new value in each cycle, an edge-triggered model cannot serve as a solution.
See the PLCOpen standard document "Creating PLCopen compliant Function Block libraries" for details.

Variant, abort used?, timeLimit, timeout, Behavior
ETrig,       FALSE,       0,        0,    Base: activates on front, ends on readyCondition
ETrigTo,     FALSE,       0,        > 0,  With timeout: if it doesn't finish within timeout, it goes to Error.
ETrigTI,     FALSE,       > 0,      0,    With timeLimit: allows you to divide the work over multiple cycles.
ETrigTITo,   FALSE,       > 0,      > 0,  Complete: both cyclical limit and total timeout management.
ETrigA,      TRUE,        0,        0,    With Aborting: It can be stopped and switched to Aborted.
ETrigATo,    TRUE,        0,        > 0,  With Aborting and timeout: if it doesn't finish within timeout, it goes to Error.
ETrigATI,    TRUE,        > 0,      0,    With Aborting and timeLimit: allows you to divide the work over multiple cycles.
ETrigATITo,  TRUE,        > 0,      > 0,  Complete: both Aborting, cyclical limit and total timeout management.

*)
FUNCTION_BLOCK EdgeTrigStatusMgr
VAR_INPUT
	(* Initialize and start operation on rising edge and stay active till finalized or aborted. *)
    execute : BOOL;
    readyCondition : BOOL; (* Operation completed feedback *)
	(* Interrupt request (ETrigA Variants) to abort the process. *)
    abortRequest : BOOL;
    abortComplete : BOOL; (* Aborting feedback *)
    resetRequest : BOOL; (* Manual reset request *)
    resetComplete : BOOL; (* Reset feedback *)
    errorCondition : BOOL; (* Functional error from external logic *)
	(*
	 * PLCOpen: timeLimit (Tl): here the time limit is set that
	 * the operation stays within the cycle time.
	 * In that way a longer operation can be divided over several cycles.
	 *)
    timeLimit : UINT; (* 0 = inactive *)
	(*
     * PLCOpen: timeout (To): the overall operating time of the
	 * defined operation should be lower than the time(in μs)
     * as specified by the input value timeout.
	 * The combination of them both (TlTo) is valid.
     *)
    timeout : UINT; (* 0 = inactive *)
    clock : BOOL; (* Clock signal *)
END_VAR
VAR_OUTPUT
    done : BOOL; (* Operation completed successfully *)
    busy : BOOL; (* Operation in progress *)
    error : BOOL; (* Active error *)
    errorId : INT; (* PLCopen: Error ID. Example 1 = ExternalError, 2 = Timeout *)
    aborted : BOOL; (* Operation aborted *)
    activeCycle : BOOL; (* TRUE when the caller needs to execute the logic *)
END_VAR
VAR
    status : EdgeTriggerStatus := EdgeTriggerStatus.Dormant; (* FSM internal status. States: 0- Dormant, 1 - Executing, 2 - Done, 3 - Aborting, 4 - Aborted, 5 - Resetting, 6 - Error *)
    timeLimitTimer : UINT;
    timeoutTimer : UINT;
    prevExecute : BOOL; (* Memory for edge detection *)
END_VAR

(*#-#-#-#-#-#-#-#-#-#---Implementation---#-#-#-#-#-#-#-#-#-#-#-#-#*)

(* Time management *)
IF clock THEN
	(* TimeLimit (Tl): cyclic timeslice management *)
	IF timeLimit > 0 AND status = EdgeTriggerStatus.Executing THEN
		IF timeLimitTimer > 0 THEN
			timeLimitTimer := timeLimitTimer - 1;
		ELSE
			(* New invocation timeslice *)
			timeLimitTimer := timeLimit;
		END_IF;
	END_IF;

	(* TimeOut (To): The total timeout only runs during execution *)
	IF timeoutTimer > 0 AND status = EdgeTriggerStatus.Executing THEN
		timeoutTimer := timeoutTimer - 1;
	END_IF;
END_IF;

CASE status OF
    EdgeTriggerStatus.Dormant :
        done := FALSE; busy := FALSE; aborted := FALSE; error := FALSE; errorId := 0; activeCycle := FALSE;

        (* Rising edge detection *)
        IF execute AND NOT prevExecute THEN
            timeoutTimer := timeout;
			timeLimitTimer := timeLimit;
            status := EdgeTriggerStatus.Executing;
        END_IF;

    EdgeTriggerStatus.Executing :
        busy := TRUE;
		(* Enable caller logic: active if there is no cycle limit or if the cycle time has not expired. *)
        activeCycle := (timeLimit = 0) OR (timeLimitTimer > 0);

        IF errorCondition OR ((timeout > 0) AND (timeoutTimer = 0)) THEN
            status := EdgeTriggerStatus.Error;
        ELSIF abortRequest THEN
            status := EdgeTriggerStatus.Aborting;
        ELSIF readyCondition THEN
            status := EdgeTriggerStatus.Done; (* Target achieved *)
        END_IF;

    EdgeTriggerStatus.Aborting :
        activeCycle := FALSE;

        IF errorCondition OR ((timeout > 0) AND (timeoutTimer = 0)) THEN
            status := EdgeTriggerStatus.Error;
        ELSIF abortComplete THEN
			status := EdgeTriggerStatus.Aborted;
		END_IF;

    EdgeTriggerStatus.Aborted :
        busy := FALSE; aborted := TRUE;

        (* Transition to resetting on the falling edge of execute *)
        IF resetRequest OR NOT execute THEN
			status := EdgeTriggerStatus.Resetting;
		END_IF;

    EdgeTriggerStatus.Done :
        busy := FALSE; done := TRUE; activeCycle := FALSE;

		(* Transition to resetting on the falling edge of execute *)
        IF resetRequest OR NOT execute THEN
			status := EdgeTriggerStatus.Resetting;
		END_IF;

    EdgeTriggerStatus.Error :
        busy := FALSE; activeCycle := FALSE; error := TRUE;

        IF errorCondition THEN
            errorId := 1; (* ExternalError *)
        ELSE
            errorId := 2; (* Total timeout expired *)
        END_IF;

        IF resetRequest OR NOT execute THEN
			status := EdgeTriggerStatus.Resetting;
		END_IF;

    EdgeTriggerStatus.Resetting :
        done := FALSE; aborted := FALSE; error := FALSE; errorId := 0; activeCycle := FALSE;

		IF resetComplete THEN
			status := EdgeTriggerStatus.Dormant;
		END_IF;
END_CASE;

prevExecute := execute;

(* ---- EdgeTrigStatusMgr.st ---- *)
(*
Edge triggered status manager.
The PLCOpen standard presents "service/command" function block patterns
that manage the execution of a request (edge-triggered)
or the maintenance of a condition (level-controlled).
The PLCopen patterns model the lifecycle of a command, not the state of the device.
A command handler FB uses the PLCopen (Action) pattern.
The device model maintains the bistable state (Reality/Feedback).
The command requests a device transition, but does not define the device state.
It makes sense to model triggers and levels for physical devices only as an interface contract
between the caller and the device controller, not as the "physical truth" of the device.
An example of edge-triggered functionality is a move-to-position command which,
after being initialized via the input execute, runs till finalized.
For the detection of a rising edge in a function block, two PLC cycles are necessary.
Thus, if the requirement is to be able to process a new value in each cycle, an edge-triggered model cannot serve as a solution.
See the PLCOpen standard document "Creating PLCopen compliant Function Block libraries" for details.

Variant, abort used?, timeLimit, timeout, Behavior
ETrig,       FALSE,       0,        0,    Base: activates on front, ends on readyCondition
ETrigTo,     FALSE,       0,        > 0,  With timeout: if it doesn't finish within timeout, it goes to Error.
ETrigTI,     FALSE,       > 0,      0,    With timeLimit: allows you to divide the work over multiple cycles.
ETrigTITo,   FALSE,       > 0,      > 0,  Complete: both cyclical limit and total timeout management.
ETrigA,      TRUE,        0,        0,    With Aborting: It can be stopped and switched to Aborted.
ETrigATo,    TRUE,        0,        > 0,  With Aborting and timeout: if it doesn't finish within timeout, it goes to Error.
ETrigATI,    TRUE,        > 0,      0,    With Aborting and timeLimit: allows you to divide the work over multiple cycles.
ETrigATITo,  TRUE,        > 0,      > 0,  Complete: both Aborting, cyclical limit and total timeout management.

*)
FUNCTION_BLOCK EdgeTrigStatusMgr
	VAR_INPUT
		(* Initialize and start operation on rising edge and stay active till finalized or aborted. *)
	    execute : BOOL;
	    readyCondition : BOOL; (* Operation completed feedback *)
		(* Interrupt request (ETrigA Variants) to abort the process. *)
	    abortRequest : BOOL;
	    abortComplete : BOOL; (* Aborting feedback *)
	    resetRequest : BOOL; (* Manual reset request *)
	    resetComplete : BOOL; (* Reset feedback *)
	    errorCondition : BOOL; (* Functional error from external logic *)
		(*
		 * PLCOpen: timeLimit (Tl): here the time limit is set that
		 * the operation stays within the cycle time.
		 * In that way a longer operation can be divided over several cycles.
		 *)
	    timeLimit : UINT; (* 0 = inactive *)
		(*
	     * PLCOpen: timeout (To): the overall operating time of the
		 * defined operation should be lower than the time(in μs)
	     * as specified by the input value timeout.
		 * The combination of them both (TlTo) is valid.
	     *)
	    timeout : UINT; (* 0 = inactive *)
	    clock : BOOL; (* Clock signal *)
	END_VAR
	VAR_OUTPUT
	    done : BOOL; (* Operation completed successfully *)
	    busy : BOOL; (* Operation in progress *)
	    error : BOOL; (* Active error *)
	    errorId : INT; (* PLCopen: Error ID. Example 1 = ExternalError, 2 = Timeout *)
	    aborted : BOOL; (* Operation aborted *)
	    activeCycle : BOOL; (* TRUE when the caller needs to execute the logic *)
	END_VAR
	VAR
	    status : EdgeTriggerStatus := EdgeTriggerStatus.Dormant; (* FSM internal status. States: 0- Dormant, 1 - Executing, 2 - Done, 3 - Aborting, 4 - Aborted, 5 - Resetting, 6 - Error *)
	    timeLimitTimer : UINT;
	    timeoutTimer : UINT;
	    prevExecute : BOOL; (* Memory for edge detection *)
	END_VAR

	(* Time management *)
	IF clock THEN
		(* TimeLimit (Tl): cyclic timeslice management *)
		IF timeLimit > 0 AND status = EdgeTriggerStatus.Executing THEN
			IF timeLimitTimer > 0 THEN
				timeLimitTimer := timeLimitTimer - 1;
			ELSE
				(* New invocation timeslice *)
				timeLimitTimer := timeLimit;
			END_IF;
		END_IF;

		(* TimeOut (To): The total timeout only runs during execution *)
		IF timeoutTimer > 0 AND status = EdgeTriggerStatus.Executing THEN
			timeoutTimer := timeoutTimer - 1;
		END_IF;
	END_IF;

	CASE status OF
	    EdgeTriggerStatus.Dormant :
	        done := FALSE; busy := FALSE; aborted := FALSE; error := FALSE; errorId := 0; activeCycle := FALSE;

	        (* Rising edge detection *)
	        IF execute AND NOT prevExecute THEN
	            timeoutTimer := timeout;
				timeLimitTimer := timeLimit;
	            status := EdgeTriggerStatus.Executing;
	        END_IF;

	    EdgeTriggerStatus.Executing :
	        busy := TRUE;
			(* Enable caller logic: active if there is no cycle limit or if the cycle time has not expired. *)
	        activeCycle := (timeLimit = 0) OR (timeLimitTimer > 0);

	        IF errorCondition OR ((timeout > 0) AND (timeoutTimer = 0)) THEN
	            status := EdgeTriggerStatus.Error;
	        ELSIF abortRequest THEN
	            status := EdgeTriggerStatus.Aborting;
	        ELSIF readyCondition THEN
	            status := EdgeTriggerStatus.Done; (* Target achieved *)
	        END_IF;

	    EdgeTriggerStatus.Aborting :
	        activeCycle := FALSE;

	        IF errorCondition OR ((timeout > 0) AND (timeoutTimer = 0)) THEN
	            status := EdgeTriggerStatus.Error;
	        ELSIF abortComplete THEN
				status := EdgeTriggerStatus.Aborted;
			END_IF;

	    EdgeTriggerStatus.Aborted :
	        busy := FALSE; aborted := TRUE;

	        (* Transition to resetting on the falling edge of execute *)
	        IF resetRequest OR NOT execute THEN
				status := EdgeTriggerStatus.Resetting;
			END_IF;

	    EdgeTriggerStatus.Done :
	        busy := FALSE; done := TRUE; activeCycle := FALSE;

			(* Transition to resetting on the falling edge of execute *)
	        IF resetRequest OR NOT execute THEN
				status := EdgeTriggerStatus.Resetting;
			END_IF;

	    EdgeTriggerStatus.Error :
	        busy := FALSE; activeCycle := FALSE; error := TRUE;

	        IF errorCondition THEN
	            errorId := 1; (* ExternalError *)
	        ELSE
	            errorId := 2; (* Total timeout expired *)
	        END_IF;

	        IF resetRequest OR NOT execute THEN
				status := EdgeTriggerStatus.Resetting;
			END_IF;

	    EdgeTriggerStatus.Resetting :
	        done := FALSE; aborted := FALSE; error := FALSE; errorId := 0; activeCycle := FALSE;

			IF resetComplete THEN
				status := EdgeTriggerStatus.Dormant;
			END_IF;
	END_CASE;

	prevExecute := execute;
	END_FUNCTION_BLOCK

(* ---- LevelCtrlStatusMgr.pou ---- *)
(*#-#-#-#-#-#-#-#-#-#---Declaration---#-#-#-#-#-#-#-#-#-#-#-#-#*)

{attribute 'no_assign'}
(*
Level controlled status manager.
The PLCOpen standard presents “service/command” function block patterns
that manage the execution of a request (edge-triggered)
or the maintenance of a condition (level-controlled).
The PLCopen patterns model the lifecycle of a command, not the state of the device.
A command handler FB uses the PLCopen (Action) pattern.
The device model maintains the bistable state (Reality/Feedback).
The command requests a device transition, but does not define the device state.
It makes sense to model triggers and levels for physical devices only as an interface contract
between the caller and the device controller, not as the “physical truth” of the device.
An example of a level triggered functionality is a PowerOn function,
where the power is switched on as long as the relevant input enable is set.
For the detection of a level in a function block, one PLC cycle is necessary.
Thus, if the requirement is to be able to process a new value in each cycle,
a level-controlled function block model is the preferred way to implement the required functionality.
See the PLCOpen standard document "Creating PLCopen compliant Function Block libraries" for details.

Variant, isContinuous, timeLimit, timeout, Behavior
LCon,       FALSE,         0,       0,     Base: Switch to Done when readyCondition is TRUE.
LConTo,     FALSE,         0,       > 0,   Monitors total time; errors if exceeded.
LConTI,     FALSE,         > 0,     0,     Split logic across multiple loops using activeCycle.
LConTITo,   FALSE,         > 0,     > 0,   Complete combination of cyclic time limit and total timeout.
LConC,      TRUE,          0,       0,     Continuous behaviour: Never goes to Done, ignores readyCondition.
LConTIC,    TRUE,          > 0,     0,     Continuous behaviour with cycle time management for heavy tasks.

Example of use:
	FUNCTION_BLOCK CilinderCmd
	VAR_EXTERNAL
		clks : Clocks;
	END_VAR
	VAR_INPUT
		enable : BOOL;
		timeout : UINT := 100;
		clock : BOOL;
		sensorOpened : BOOL; (* Limit switch sensor open *)
		sensorClosed : BOOL; (* Limit switch sensor closed *)
	END_VAR
	VAR_OUTPUT
		valveCmd : BOOL; (* Solenoid valve control *)
		fault : BOOL;
	END_VAR
	VAR
		(* Composition: PLCopen status manager instance *)
		statusMgr : LevelCtrlStatusMgr;
	END_VAR

	(* Sensor feedback mapping *)
	(* The cylinder is ready when the opening sensor is active *)
	statusMgr.readyCondition := sensorOpened AND NOT sensorClosed;
	(* Suppose that reset and abort are instantaneous for a cylinder *)
	statusMgr.abortComplete := TRUE;
	statusMgr.resetComplete := sensorClosed;

	statusMgr(enable := enable, timeLimit := 1, (* Example: 10 ms or 1 clock10ms pulse per cycle *)
		timeout := timeout, clock := clks.clock10ms);

	(* Physical action: based on manager's signals *)
	(* The command to the valve is given only if the manager is running *)
	IF statusMgr.activeCycle THEN
		valveCmd := TRUE;
	ELSE
		valveCmd := FALSE;
	END_IF;

	(* Diagnostics *)
	fault := statusMgr.error;

	END_FUNCTION_BLOCK
*)
FUNCTION_BLOCK LevelCtrlStatusMgr
VAR_INPUT
	(*
	 * Active while high.
     * Enable is a safety/permission condition (if it disappears, you must disable immediately),
	 * for a “fail-safe” behavior: if the caller loses enable → go to disable.
     *)
    enable : BOOL;
    readyCondition : BOOL; (* Operation completed feedback *)
    abortComplete : BOOL; (* Aborting feedback *)
    resetRequest : BOOL; (* Manual reset request *)
    resetComplete : BOOL; (* Reset feedback *)
    errorCondition : BOOL; (* Functional error from external logic *)
	(*
	 * TRUE for LConC / LConTIC variants (without Done state).
	 * PLCOpen: For continuous behaviour, meaning it does not stop
     * so there is no Done state. See the 2 additional blocks LConC
     * and LConTlC, including the time limit, for continuous behaviour.
     *)
    isContinuous : BOOL;
    (*
	 * PLCOpen: timeLimit (Tl): here the time limit is set that
	 * the operation stays within the cycle time.
	 * In that way a longer operation can be divided over several cycles.
	 *)
    timeLimit : UINT; (* 0 = inactive *)
	(*
     * PLCOpen: timeout (To): the overall operating time of the
	 * defined operation should be lower than the time(in μs)
     * as specified by the input value timeout.
	 * The combination of them both (TlTo) is valid.
     *)
    timeout : UINT; (* 0 = inactive *)
    clock : BOOL; (* Clock signal *)
END_VAR
VAR_OUTPUT
    done : BOOL; (* Operation valid / Final state reached (only if NOT isContinuous) *)
    busy : BOOL; (* Operation in progress *)
    error : BOOL; (* Active error *)
    errorId : INT; (* PLCopen: Error ID. Example 1 = Timeout *)
    activeCycle : BOOL; (* TRUE when the caller needs to execute the logic *)
END_VAR
VAR
    status : LevelCtrlStatus := LevelCtrlStatus.Dormant; (* FSM internal status. States: 0 - Dormant, 1 - Executing , 2 - Done, 3 - Aborting, 4 - Resetting, 5 - Error *)
    timeLimitTimer : UINT;
    timeoutTimer : UINT;
END_VAR

(*#-#-#-#-#-#-#-#-#-#---Implementation---#-#-#-#-#-#-#-#-#-#-#-#-#*)

(* Time management *)
IF clock THEN
	(* TimeLimit (Tl): cyclic timeslice management *)
	IF timeLimit > 0 AND status = LevelCtrlStatus.Executing THEN
		IF timeLimitTimer > 0 THEN
			timeLimitTimer := timeLimitTimer - 1;
		ELSE
			(* New invocation timeslice *)
			timeLimitTimer := timeLimit;
		END_IF;
	END_IF;

	(* TimeOut (To): The total timeout only runs during execution *)
	IF timeoutTimer > 0 AND status = LevelCtrlStatus.Executing THEN
		timeoutTimer := timeoutTimer - 1;
	END_IF;
END_IF;

CASE status OF
    LevelCtrlStatus.Dormant :
        done := FALSE; busy := FALSE; error := FALSE; errorId := 0; activeCycle := FALSE;

		(* Level detection *)
        IF enable THEN
            timeoutTimer := timeout;
			timeLimitTimer := timeLimit;
            status := LevelCtrlStatus.Executing;
        END_IF;

    LevelCtrlStatus.Executing :
        busy := TRUE;
        (* Enable caller logic: active if there is no cycle limit or if the cycle time has not expired. *)
        activeCycle := (timeLimit = 0) OR (timeLimitTimer > 0);

        IF errorCondition OR ((timeout > 0) AND (timeoutTimer = 0)) THEN
            status := LevelCtrlStatus.Error;
        ELSIF NOT enable THEN
            status := LevelCtrlStatus.Aborting;
        ELSIF NOT isContinuous AND readyCondition THEN
            status := LevelCtrlStatus.Done; (* Target achieved (Standard variants) *)
        END_IF;

    LevelCtrlStatus.Aborting :
        activeCycle := FALSE;

        IF errorCondition OR ((timeout > 0) AND (timeoutTimer = 0)) THEN
            status := LevelCtrlStatus.Error;
		ELSIF abortComplete THEN
			status := LevelCtrlStatus.Resetting;
		END_IF;

    LevelCtrlStatus.Done : (* Only for non-continuous variants *)
        busy := FALSE; done := TRUE; activeCycle := FALSE;

        IF NOT enable THEN
			status := LevelCtrlStatus.Resetting;
		END_IF;

    LevelCtrlStatus.Error :
        busy := FALSE; activeCycle := FALSE; error := TRUE;

        IF errorCondition THEN
            errorId := 1; (* ExternalError *)
        ELSE
            errorId := 2; (* Total timeout expired *)
        END_IF;

		IF resetRequest OR NOT enable THEN
			status := LevelCtrlStatus.Resetting;
		END_IF;

    LevelCtrlStatus.Resetting :
        done := FALSE; error := FALSE; errorId := 0; activeCycle := FALSE;

        IF resetComplete THEN
			status := LevelCtrlStatus.Dormant;
		END_IF;
END_CASE;

(* ---- LevelCtrlStatusMgr.st ---- *)
(*
Level controlled status manager.
The PLCOpen standard presents "service/command" function block patterns
that manage the execution of a request (edge-triggered)
or the maintenance of a condition (level-controlled).
The PLCopen patterns model the lifecycle of a command, not the state of the device.
A command handler FB uses the PLCopen (Action) pattern.
The device model maintains the bistable state (Reality/Feedback).
The command requests a device transition, but does not define the device state.
It makes sense to model triggers and levels for physical devices only as an interface contract
between the caller and the device controller, not as the "physical truth" of the device.
An example of a level triggered functionality is a PowerOn function,
where the power is switched on as long as the relevant input enable is set.
For the detection of a level in a function block, one PLC cycle is necessary.
Thus, if the requirement is to be able to process a new value in each cycle,
a level-controlled function block model is the preferred way to implement the required functionality.
See the PLCOpen standard document "Creating PLCopen compliant Function Block libraries" for details.

Variant, isContinuous, timeLimit, timeout, Behavior
LCon,       FALSE,         0,       0,     Base: Switch to Done when readyCondition is TRUE.
LConTo,     FALSE,         0,       > 0,   Monitors total time; errors if exceeded.
LConTI,     FALSE,         > 0,     0,     Split logic across multiple loops using activeCycle.
LConTITo,   FALSE,         > 0,     > 0,   Complete combination of cyclic time limit and total timeout.
LConC,      TRUE,          0,       0,     Continuous behaviour: Never goes to Done, ignores readyCondition.
LConTIC,    TRUE,          > 0,     0,     Continuous behaviour with cycle time management for heavy tasks.

Example of use:
	FUNCTION_BLOCK CilinderCmd
	VAR_EXTERNAL
		clks : Clocks;
	END_VAR
	VAR_INPUT
		enable : BOOL;
		timeout : UINT := 100;
		clock : BOOL;
		sensorOpened : BOOL; (* Limit switch sensor open *)
		sensorClosed : BOOL; (* Limit switch sensor closed *)
	END_VAR
	VAR_OUTPUT
		valveCmd : BOOL; (* Solenoid valve control *)
		fault : BOOL;
	END_VAR
	VAR
		(* Composition: PLCopen status manager instance *)
		statusMgr : LevelCtrlStatusMgr;
	END_VAR

	(* Sensor feedback mapping *)
	(* The cylinder is ready when the opening sensor is active *)
	statusMgr.readyCondition := sensorOpened AND NOT sensorClosed;
	(* Suppose that reset and abort are instantaneous for a cylinder *)
	statusMgr.abortComplete := TRUE;
	statusMgr.resetComplete := sensorClosed;

	statusMgr(enable := enable, timeLimit := 1, (* Example: 10 ms or 1 clock10ms pulse per cycle *)
		timeout := timeout, clock := clks.clock10ms);

	(* Physical action: based on manager's signals *)
	(* The command to the valve is given only if the manager is running *)
	IF statusMgr.activeCycle THEN
		valveCmd := TRUE;
	ELSE
		valveCmd := FALSE;
	END_IF;

	(* Diagnostics *)
	fault := statusMgr.error;

	END_FUNCTION_BLOCK
*)
FUNCTION_BLOCK LevelCtrlStatusMgr
VAR_INPUT
	(*
	 * Active while high.
     * Enable is a safety/permission condition (if it disappears, you must disable immediately),
	 * for a "fail-safe" behavior: if the caller loses enable -> go to disable.
     *)
    enable : BOOL;
    readyCondition : BOOL; (* Operation completed feedback *)
    abortComplete : BOOL; (* Aborting feedback *)
    resetRequest : BOOL; (* Manual reset request *)
    resetComplete : BOOL; (* Reset feedback *)
    errorCondition : BOOL; (* Functional error from external logic *)
	(*
	 * TRUE for LConC / LConTIC variants (without Done state).
	 * PLCOpen: For continuous behaviour, meaning it does not stop
     * so there is no Done state. See the 2 additional blocks LConC
     * and LConTlC, including the time limit, for continuous behaviour.
     *)
    isContinuous : BOOL;
    (*
	 * PLCOpen: timeLimit (Tl): here the time limit is set that
	 * the operation stays within the cycle time.
	 * In that way a longer operation can be divided over several cycles.
	 *)
    timeLimit : UINT; (* 0 = inactive *)
	(*
     * PLCOpen: timeout (To): the overall operating time of the
	 * defined operation should be lower than the time(in μs)
     * as specified by the input value timeout.
	 * The combination of them both (TlTo) is valid.
     *)
    timeout : UINT; (* 0 = inactive *)
    clock : BOOL; (* Clock signal *)
END_VAR
VAR_OUTPUT
    done : BOOL; (* Operation valid / Final state reached (only if NOT isContinuous) *)
    busy : BOOL; (* Operation in progress *)
    error : BOOL; (* Active error *)
    errorId : INT; (* PLCopen: Error ID. Example 1 = Timeout *)
    activeCycle : BOOL; (* TRUE when the caller needs to execute the logic *)
END_VAR
VAR
    status : LevelCtrlStatus := LevelCtrlStatus.Dormant; (* FSM internal status. States: 0 - Dormant, 1 - Executing , 2 - Done, 3 - Aborting, 4 - Resetting, 5 - Error *)
    timeLimitTimer : UINT;
    timeoutTimer : UINT;
END_VAR

(* Time management *)
IF clock THEN
	(* TimeLimit (Tl): cyclic timeslice management *)
	IF timeLimit > 0 AND status = LevelCtrlStatus.Executing THEN
		IF timeLimitTimer > 0 THEN
			timeLimitTimer := timeLimitTimer - 1;
		ELSE
			(* New invocation timeslice *)
			timeLimitTimer := timeLimit;
		END_IF;
	END_IF;

	(* TimeOut (To): The total timeout only runs during execution *)
	IF timeoutTimer > 0 AND status = LevelCtrlStatus.Executing THEN
		timeoutTimer := timeoutTimer - 1;
	END_IF;
END_IF;

CASE status OF
    LevelCtrlStatus.Dormant :
        done := FALSE; busy := FALSE; error := FALSE; errorId := 0; activeCycle := FALSE;

		(* Level detection *)
        IF enable THEN
            timeoutTimer := timeout;
			timeLimitTimer := timeLimit;
            status := LevelCtrlStatus.Executing;
        END_IF;

    LevelCtrlStatus.Executing :
        busy := TRUE;
        (* Enable caller logic: active if there is no cycle limit or if the cycle time has not expired. *)
        activeCycle := (timeLimit = 0) OR (timeLimitTimer > 0);

        IF errorCondition OR ((timeout > 0) AND (timeoutTimer = 0)) THEN
            status := LevelCtrlStatus.Error;
        ELSIF NOT enable THEN
            status := LevelCtrlStatus.Aborting;
        ELSIF NOT isContinuous AND readyCondition THEN
            status := LevelCtrlStatus.Done; (* Target achieved (Standard variants) *)
        END_IF;

    LevelCtrlStatus.Aborting :
        activeCycle := FALSE;

        IF errorCondition OR ((timeout > 0) AND (timeoutTimer = 0)) THEN
            status := LevelCtrlStatus.Error;
		ELSIF abortComplete THEN
			status := LevelCtrlStatus.Resetting;
		END_IF;

    LevelCtrlStatus.Done : (* Only for non-continuous variants *)
        busy := FALSE; done := TRUE; activeCycle := FALSE;

        IF NOT enable THEN
			status := LevelCtrlStatus.Resetting;
		END_IF;

    LevelCtrlStatus.Error :
        busy := FALSE; activeCycle := FALSE; error := TRUE;

        IF errorCondition THEN
            errorId := 1; (* ExternalError *)
        ELSE
            errorId := 2; (* Total timeout expired *)
        END_IF;

		IF resetRequest OR NOT enable THEN
			status := LevelCtrlStatus.Resetting;
		END_IF;

    LevelCtrlStatus.Resetting :
        done := FALSE; error := FALSE; errorId := 0; activeCycle := FALSE;

        IF resetComplete THEN
			status := LevelCtrlStatus.Dormant;
		END_IF;
END_CASE;

(* ---- ProcessPid.pou ---- *)
(*#-#-#-#-#-#-#-#-#-#---Declaration---#-#-#-#-#-#-#-#-#-#-#-#-#*)

{attribute 'no_assign'}
(* Process PID *)
FUNCTION_BLOCK ProcessPid
VAR_INPUT
    enable : BOOL; (* Master enable: if FALSE, resets the PID and clears the outputs *)
    reset : BOOL; (* Manual reset of internal components *)
    (* Control system metadata for logging purpose *)
    controlSystemId : STRING;
    controlSystemName : STRING;
    (* The actual value of process feedback *)
    feedback : REAL;
    (* Defines the multiplier with which the feedback is multiplied *)
    feedbackMultiplier : REAL := 1.0;
    (* Setpoint. The running direction for the setpoint is determined by the sign of the setpoint itself. *)
    setpoint : REAL;
    (* Defines the “at setpoint” limits for output control of the device.
     * When the difference between the setpoint and the feedback is smaller than this hysteresis,
     * the device is considered to be “at setpoint”.
     *)
    atSetpointHysteresis : REAL;
    (* Defines the multiplier with which the setpoint is multiplied *)
    setpointMultiplier : REAL := 1.0;
    (* Defines a minimum limit for the process PID controller setpoint *)
    setpointMin : REAL;
    (* Defines a maximum limit for the process PID controller setpoint *)
    setpointMax : REAL;
    (* Select a ramp function to increase the setpoint *)
    setpointRampType : RampType := RampType.Linear;
    (* Defines the minimum time it takes for the setpoint to increase from 0% to 100% *)
    setpointIncreaseTime : TIME := T#0S;
    (* Defines the minimum time it takes for the setpoint to decrease from 100% to 0% *)
    setpointDecreaseTime : TIME := T#0S;
    (* Freezes the setpoint of the process PID controller *)
    setpointFreezeEnable : BOOL;
    (* Inverts the input of the process PID controller.
     * Deviation not inverted (Deviation = Setpoint - Feedback).
     * Deviation inverted (Deviation = Feedback - Setpoint).
     *)
    deviationInversion : BOOL;
    (* Defines the minimum limit for the process PID controller output. Using the minimum and maximum limits, it is possible to restrict the operation range *)
    outputMin : REAL;
    (* Defines the maximum limit for the process PID controller output *)
    outputMax : REAL;
    (* Freezes (or defines a source that can be used to freeze) the output of the process PID controller, keeping the output at the value it was before freeze was enabled.
     * This feature can be used when, for example, a sensor providing process feedback must to be serviced without stopping the process.
     *)
    outputFreezeEnable : BOOL;
    (* Defines the gain for the process PID controller *)
    gain : REAL := 1.0;
    (* Defines the integration time for the process PID controller.
     * This time needs to be set to the same order of magnitude as
     * the reaction time of the process being controlled, otherwise
     * instability will result.
     *)
    integrationTime : REAL := 0.0;
    (* The derivative component. Defines the derivation time of the process PID controller. *)
    derivationTime : REAL := 0.0;
    (* Offset for the output variable *)
    offset : REAL := 0.0;
    (* Defines a deadband around the setpoint.
     * Whenever process feedback enters the deadband, a delay timer starts.
     * If the feedback remains within the deadband longer than the delay (set deadband delay),
     * the PID controller output is frozen. Normal operation resumes after the feedback value leaves the deadband.
     *)
    deadbandRange : REAL;
    (* Delay for the deadband *)
    deadbandDelay : TIME;
    (* Defines the start limit for the sleep function. If the value is 0.0, set 1 sleep mode is disabled.
     * The sleep function compares PID output (parameter PID output actual) to the value of this parameter.
     * If PID output remains below this value longer than the sleep delay,
     * the drive enters the sleep mode and stops the motor. If the value is 0.0, sleep mode is disabled.
     *)
    sleepLevel : REAL := 0.0;
    (* Defines a delay before the sleep function actually becomes enabled,
     * to prevent nuisance sleeping. The delay timer starts when the sleep mode is enabled by
     * parameter sleep level, and resets when the sleep mode is disabled.
     *)
    sleepDelay : TIME;
    (* Defines the wake-up level as deviation between process setpoint and feedback.
     * When the deviation exceeds the value of this parameter, and remains there for
     * the duration of the wake-up delay, the drive wakes up.
     *)
    wakeupDeviation : REAL;
    (* Defines a wake-up delay for the sleep function to prevent nuisance wake-ups.
     * The delay timer starts when the deviation exceeds the wake-up level (wake-up deviation),
     * and resets if the deviation falls below the wake-up level.
     *)
    wakeupDelay : TIME;
    (* Defines the output level forced during the sleep boost phase.
     * If 0.0 or sleepBoostTime is T#0S, the boost phase is skipped and sleep is entered directly.
     *)
    sleepBoostLevel : REAL := 0.0;
    (* Defines how long the output is held at sleepBoostLevel before entering sleep mode. *)
    sleepBoostTime : TIME;
    (* Activates (or selects a source that activates) tracking mode.
     * In tracking mode, the value selected by parameter tracking reference is substituted for the PID controller output.
     *)
    trackingMode : BOOL := FALSE;
    trackingRef : REAL := 0.0;
    (* Timing *)
    clock : BOOL; (* Tick pulse, e.g. clks.clock10ms *)
    tickTime : TIME := T#10ms;
    (* Optional setpoint change epsilon (avoid restart on tiny changes) *)
    setpointEpsilon : REAL := 0.000001;
END_VAR
(* Process PID outputs and diagnostics *)
VAR_OUTPUT
    (* Displays the value of process PID feedback after processing *)
    feedbackActual : REAL;
    (* Displays the value of process PID setpoint after processing *)
    setpointActual : REAL;
    (* Displays the process PID deviation. By default, this value equals setpoint - feedback, but deviation can be inverted by parameter deviationInversion. *)
    deviationActual : REAL;
    (* Displays the output of the controller *)
    outputActual : REAL;
    (* Diagnostics. It display status information on process PID control. *)
    invalidConfig : BOOL;
    active, (* Indicates that the process PID has control on the device *)
    atSetpoint, (* The device is at setpoint *)
    zeroOutput, (* Device is at zero output *)
    setpointFrozen, (* Process PID setpoint frozen *)
    outputFrozen, (* Process PID controller output frozen *)
    sleepMode, (* Sleep mode active *)
    sleepBoost, (* Sleep boost active: output is held at sleepBoostLevel before entering sleep mode *)
    deadband, (* Feedback value is in the deadband range *)
    tracking, (* Tracking function active *)
    outputLimitsActive, (* The output has exceeded the given limits outputMin, outputMax and is limited to these values *)
    overflow : BOOL; (* Overflow in integral part *)
    (* Logger name for the signal management *)
    loggerName : STRING;
END_VAR
VAR
    (* PID controller *)
    pid : PID;
    (* Deadband timer *)
    deadbandTimer : TON;
    (* Sleep mode timer *)
    sleepTimer : TON;
    (* Sleep boost timer *)
    sleepBoostTimer : TON;
    (* Wake-up timer *)
    wakeupTimer : TON;
    (* Internal setpoint and output *)
    setpointTarget : REAL;
    setpointInternal : REAL;
    (* Last setpoint value *)
    lastSetpoint : REAL;
    lastSetpointTarget : REAL;
    outputInternal : REAL;
    (* Last output value *)
    lastOutput : REAL;
    (* For sleep decision (use last PID output to avoid cyclic dependency) *)
    lastPidOutput : REAL;
    (* Internal execution control *)
    execute : BOOL;
    manualMode : BOOL;
    yManual : REAL;
    sleepReq : BOOL;
    wakeupReq : BOOL;
    (* Reset edge handling *)
    prevReset : BOOL;
    resetEdge : BOOL;
    (* Ramp generator *)
    rampFunc : RAMP_REAL;
    (* S-shaped function *)
    sShapedFunc : SShapedFunc;
    (* Exponential ramp helper (uses time constant in seconds) *)
    expRamp : IIRFilter;
    (* Ramp helpers *)
    incMs, decMs : DINT;
    incSec, decSec, spRange, ascRate, decRate : REAL;
    (* Ramp (S-shaped / exponential) start *)
    startRamp : BOOL;
    expTau : REAL;
    (* Logger facade *)
    logger : LoggerFacade;
END_VAR

(*#-#-#-#-#-#-#-#-#-#---Implementation---#-#-#-#-#-#-#-#-#-#-#-#-#*)

(* Master enable gate *)
IF NOT enable THEN
    (* If disabled, force resets and clear all outputs to zero *)
    active := FALSE;
    execute := FALSE;
    outputActual := 0.0;
    zeroOutput := TRUE;
    atSetpoint := FALSE;

    (* Reset internal asynchronous components to prevent wind-up or jumps on re-enable *)
    pid(reset := TRUE);
    rampFunc(reset := TRUE);
    deadbandTimer(IN := FALSE);
    sleepTimer(IN := FALSE);
    sleepBoostTimer(IN := FALSE);
    wakeupTimer(IN := FALSE);
    sleepMode := FALSE;
    sleepBoost := FALSE;

    RETURN; (* Stop execution *)
END_IF;

(* Args validation *)
invalidConfig := FALSE;
IF (controlSystemId = '' AND controlSystemName = '') THEN
    active := FALSE;
    execute := FALSE;
    invalidConfig := TRUE;
    RETURN;
END_IF;

(* Logger facade init *)
loggerName := concat(concat(concat(controlSystemName, '['), controlSystemId), ']');
logger.enable := TRUE; logger.loggerName := loggerName;

(* Configuration parameters validation *)
IF (integrationTime < 0) OR (derivationTime < 0) OR (gain <= 0)
        OR (setpointMin > setpointMax) OR (outputMin > outputMax) THEN
    logger(message := 'Invalid PID arguments detected.', level := LogLevel.Error);
    active := FALSE;
    execute := FALSE;
    invalidConfig := TRUE;
    RETURN;
END_IF;

(* Enable core logic *)
active := TRUE;
execute := TRUE;

logger(message := 'Running process PID.', level := LogLevel.Debug);

(* Reset handling *)
resetEdge := reset AND NOT prevReset;
prevReset := reset;

IF resetEdge THEN
    logger(message := 'Reset process PID.', level := LogLevel.Warn);
    setpointTarget := 0; setpointInternal := 0; setpointActual := 0;
    lastSetpoint := 0; lastSetpointTarget := 0;
    deviationActual := 0; outputInternal := 0; outputActual := 0;
    lastOutput := 0; lastPidOutput := 0;
    deadbandTimer(IN := FALSE); sleepTimer(IN := FALSE); sleepBoostTimer(IN := FALSE); wakeupTimer(IN := FALSE);
    rampFunc(reset := TRUE);
    sShapedFunc(execute := FALSE); expRamp(execute := FALSE, reset := TRUE);
    pid(reset := TRUE);
    sleepMode := FALSE;
    sleepBoost := FALSE;
END_IF;

(* Feedback processing (scaling) *)
feedbackActual := feedback * feedbackMultiplier;
logger(message := concat('Input feedback value ', TO_STRING(feedback)), level := LogLevel.Debug);
logger(message := concat('Scaled feedback value ', TO_STRING(feedbackActual)), level := LogLevel.Debug);

(* Setpoint processing (limit + ramp + freeze). *)
IF setpointFreezeEnable THEN
    logger(message := concat('Setpoint freezed at value', TO_STRING(lastSetpoint)), level := LogLevel.Debug);
    setpointTarget := lastSetpoint;
ELSE
    setpointTarget := LIMIT(setpointMin, setpoint * setpointMultiplier, setpointMax);
END_IF;

(* Ramp is enabled only when both times are > 0 *)
IF (setpointIncreaseTime > T#0S) AND (setpointDecreaseTime > T#0S) THEN
    logger(message := 'Setpoint ramp up enabled.', level := LogLevel.Debug);

    (* Detect target changes to restart the ramp generator (epsilon-based) *)
    startRamp := (ABS(setpointTarget - lastSetpointTarget) > setpointEpsilon) OR resetEdge;
    lastSetpointTarget := setpointTarget;

    CASE setpointRampType OF
        RampType.SShaped :
            sShapedFunc(execute := startRamp OR sShapedFunc.busy, clock := clock,
                startValue := lastSetpoint, endValue := setpointTarget,
                duration := SEL(setpointTarget >= lastSetpoint, setpointDecreaseTime, setpointIncreaseTime),
                tickTime := tickTime);
            setpointInternal := SEL(sShapedFunc.error, sShapedFunc.output, setpointTarget);

        RampType.Linear :
            incMs := TO_DINT(setpointIncreaseTime); decMs := TO_DINT(setpointDecreaseTime);
            incSec := MAX(0.001, TO_REAL(incMs) / 1000.0); decSec := MAX(0.001, TO_REAL(decMs) / 1000.0);
            spRange := MAX(1.0, setpointMax - setpointMin);
            ascRate := spRange / incSec; decRate := spRange / decSec;
            rampFunc(in := setpointTarget, ascend := ascRate, descend := decRate,
                timebase := tickTime, reset := resetEdge, out => setpointInternal);

        RampType.Exponential :
        	(*
             * Exponential ramp: use ExpFilter as a first-order approach to target.
			 * We select a time constant tau such that the response reaches ~99% at the configured ramp time.
			 * For a first-order system: 1 - exp(-t/tau) = 0.99 -> tau = t / 4.605
			 *)
            expTau := TO_REAL(TO_DINT(SEL(setpointTarget >= lastSetpoint, setpointDecreaseTime, setpointIncreaseTime))) / 4605.0; (* T / 4.605 *)
            expRamp(execute := TRUE, clock := clock, reset := startRamp, input := setpointTarget, T := MAX(0.001, expTau), tickTime := tickTime);
            setpointInternal := SEL(expRamp.error, expRamp.output, setpointTarget);
    END_CASE;
    lastSetpoint := setpointInternal;
ELSE
    setpointInternal := setpointTarget;
    lastSetpoint := setpointInternal;
    lastSetpointTarget := setpointTarget;
END_IF;

(* Update the process PID status *)
setpointFrozen := setpointFreezeEnable;
setpointActual := setpointInternal;
logger(message := concat('Actual setpoint value ', TO_STRING(setpointActual)), level := LogLevel.Debug);

(* Deviation and control modes *)
(* Deviation calculation *)
deviationActual := SEL(deviationInversion, setpointActual - feedbackActual, feedbackActual - setpointActual);
logger(message := concat('Actual deviation value ', TO_STRING(deviationActual)), level := LogLevel.Debug);

(* Deadband logic *)
deadbandTimer(IN := (deadbandRange > 0.0) AND (ABS(deviationActual) <= deadbandRange), PT := deadbandDelay);
deadband := deadbandTimer.Q;

(*
 * Sleep mode logic. Sleep enabled only when sleepLevel > 0.
 * ABB semantics: compare PID output actual to sleepLevel and wait sleepDelay.
 * We use lastPidOutput (one-cycle delayed) to avoid a cyclic dependency.
 * This is acceptable because sleep has a delay timer.
 *)
sleepReq := (sleepLevel > 0.0) AND (lastPidOutput <= sleepLevel) AND (NOT sleepMode) AND (NOT sleepBoost) AND (NOT trackingMode);
sleepTimer(IN := sleepReq, PT := sleepDelay);

(* Wake-up logic *)
wakeupReq := (wakeupDeviation > 0.0) AND (ABS(deviationActual) >= wakeupDeviation) AND sleepMode;
wakeupTimer(IN := wakeupReq, PT := wakeupDelay);

IF sleepTimer.Q THEN
    sleepTimer(IN := FALSE);
    IF (sleepBoostLevel > 0.0) AND (sleepBoostTime > T#0S) THEN
        logger(message := 'Sleep boost started.', level := LogLevel.Debug);
        sleepBoost := TRUE;
    ELSE
        logger(message := 'Sleep mode enabled.', level := LogLevel.Debug);
        sleepMode := TRUE;
    END_IF;
END_IF;

(* Sleep boost timer: hold sleepBoostLevel for sleepBoostTime, then enter sleep *)
sleepBoostTimer(IN := sleepBoost, PT := sleepBoostTime);
IF sleepBoostTimer.Q THEN
    logger(message := 'Sleep boost completed. Entering sleep mode.', level := LogLevel.Debug);
    sleepBoost := FALSE;
    sleepBoostTimer(IN := FALSE);
    sleepMode := TRUE;
END_IF;

IF wakeupTimer.Q THEN
    logger(message := 'Sleep mode disabled. Wakeup the PID.', level := LogLevel.Debug);
    sleepMode := FALSE;
    (* Reset sleep timer once awake (prevents immediate re-sleep) *)
    sleepTimer(IN := FALSE);
END_IF;

(* PID calculation and output gating *)
(* Priority (substitution/freeze functions): Tracking > SleepBoost > Sleep > Deadband > Freeze *)
tracking := FALSE; manualMode := FALSE;
yManual := lastOutput;

IF trackingMode THEN
    logger(message := 'Tracking mode enabled.', level := LogLevel.Debug);
    tracking := TRUE; manualMode := TRUE; yManual := trackingRef;
    sleepTimer(IN := FALSE);
    sleepBoost := FALSE; sleepBoostTimer(IN := FALSE);
ELSIF sleepBoost THEN
    manualMode := TRUE; yManual := sleepBoostLevel;
ELSIF sleepMode THEN
    manualMode := TRUE; yManual := 0.0;
ELSIF deadband THEN
    logger(message := 'Deadband enabled.', level := LogLevel.Debug);
    manualMode := TRUE; yManual := lastOutput;
ELSE
    manualMode := outputFreezeEnable;
    yManual := lastOutput;
END_IF;

(* Core PID execution *)
pid(actual := feedbackActual, set_point := setpointActual, kp := gain, tn := integrationTime, tv := derivationTime,
    y_manual := yManual, y_offset := offset, y_min := outputMin, y_max := outputMax,
    manual := manualMode, reset := resetEdge, y => outputInternal,
    limits_active => outputLimitsActive, overflow => overflow);

IF overflow THEN
    logger(message := 'PID overflow. Resetting the integral part.', level := LogLevel.Error);
END_IF;

IF outputLimitsActive THEN
    logger(message := 'Output limits active.', level := LogLevel.Debug);
END_IF;

(* Update ABB-like output reference for sleep decision *)
lastPidOutput := outputInternal;

(* Apply final output substitution rules consistent with selected mode *)
outputActual := outputInternal;
logger(message := concat('Actual output value ', TO_STRING(outputActual)), level := LogLevel.Debug);

outputFrozen := outputFreezeEnable OR deadband;
zeroOutput := (ABS(outputActual) < setpointEpsilon);
lastOutput := outputActual;
IF zeroOutput THEN
	logger(message := 'PID output to zero', level := LogLevel.Debug);
END_IF;

IF ABS(deviationActual) < atSetpointHysteresis THEN
		logger(message := 'PID at setpoint.', level := LogLevel.Debug);
    atSetpoint := TRUE;
ELSE
    atSetpoint := FALSE;
END_IF;
